FUNCTION_BLOCK FB_PID_Controller
VAR_INPUT
	setpoint : REAL;
	feedback : REAL;
	KP : REAL;
	KI : REAL;
	KD : REAL;
END_VAR
VAR_OUTPUT
	controlSignal : REAL;
END_VAR
VAR
	currentError : REAL;
	accumulatedError : REAL;
	deltaError : REAL;
END_VAR

error := setpoint - feedback;

controlSignal := KP*error + KI*accumulatedError + KD*deltaError;

END_FUNCTION_BLOCK

(* stored: Version 1.1.0.1, ProductVersion 3.1.4024.13
   POU FB_PID_Controller: Id {0bc8d511-12ca-4dfb-ad0e-bd1e6c62fad3}, SpecialFunc None *)
